FUNCTION_BLOCK MachineCoordinator
  (* Version 1.0, 2006-11-13, Goran Cengic, Chalmers *)
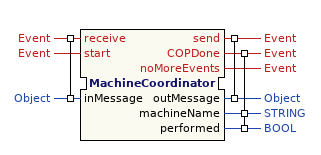
  EVENT_INPUT
    receive WITH inMessage;
    start;
  END_EVENT
  EVENT_OUTPUT
    send WITH outMessage;
    COPDone WITH machineName, performed;
    noMoreEvents;
  END_EVENT
  VAR_INPUT
    inMessage : Object;
  END_VAR
  VAR_OUTPUT
    outMessage : Object;
    machineName : STRING;
    performed : BOOL;
  END_VAR
END_FUNCTION_BLOCK
